// TIA Portal V17 export
// export: Created 2025-03-07T09:19:26.4228725Z, ExportSetting WithDefaults, DisplayName Totally Integrated Automation Portal, DisplayVersion V17 Update 8, DisplayName TIA Portal Openness, DisplayVersion V17 Update 8, DisplayName TIA Portal Version Control Interface, DisplayVersion V17, DisplayName SINAMICS Startdrive Advanced, DisplayVersion V17 SP2, DisplayName SINAMICS Startdrive G110M, G120, G120C, G120D, G120P, G115D, DisplayVersion V17 SP2, DisplayName SINAMICS Startdrive G130, G150, S120, S150, SINAMICS MV, S210, DisplayVersion V17 SP2, DisplayName STEP 7 Professional, DisplayVersion V17 Update 8, DisplayName SINUMERIK ONE STEP 7 Toolbox, DisplayVersion V17 Update 12, DisplayName SINUMERIK 840D sl STEP 7 Toolbox, DisplayVersion V17 Update 12, DisplayName STEP 7 Safety, DisplayVersion V17 Update 6, DisplayName WinCC Advanced, DisplayVersion V17 Update 8
TYPE "LBP_typeConfigData"
TITLE = Configuration parameter / Parámetros de configuración / Konfigurationsparameter
// User data type for block LBP_ConfigData [DB7] / Tipo de dato de usuario para bloque LBP_ConfigData [DB7] / Anwender-Datentyp für Baustein LBP_ConfigData [DB7]
// stored: IsFailsafeCompliant false
   STRUCT
      MCPNum : Int;   // Eingänge beginnen hier / Inputs starting here / Entradas comienzan aquí
      MCP1In : Struct   // Zeiger / Pointer / Puntero
         DBNo : Word;
         Addr : DWord;
      END_STRUCT;
      MCP1Out : Struct   // Zeiger / Pointer / Puntero
         DBNo : Word;
         Addr : DWord;
      END_STRUCT;
      reservedByte14_25 : Array[14..25] of Byte;
      MCP1BusAdr : Int := 6;
      MCP1Timeout : S5Time := S5T#700MS;
      reservedByte30_31 : Array[30..31] of Byte;
      MCP2In : Struct   // Zeiger / Pointer / Puntero
         DBNo : Word;
         Addr : DWord;
      END_STRUCT;
      MCP2Out : Struct   // Zeiger / Pointer / Puntero
         DBNo : Word;
         Addr : DWord;
      END_STRUCT;
      reservedByte44_55 : Array[44..55] of Byte;
      MCP2BusAdr : Int;
      MCP2Timeout : S5Time := S5T#700MS;
      reservedByte60_61 : Array[60..61] of Byte;
      reservedBool62_0 : Bool;
      MCP1Stop : Bool;
      MCP2Stop : Bool;
      MCP1NotSend : Bool;
      MCP2NotSend : Bool;
      reservedBool62_5 : Bool;
      reservedBool62_6 : Bool;
      MCPBusType : Byte := BYTE#16#05;
      HTIf : Int;
      HTIn : Struct   // Zeiger / Pointer / Puntero
         DBNo : Word;
         Addr : DWord;
      END_STRUCT;
      HTOut : Struct   // Zeiger / Pointer / Puntero
         DBNo : Word;
         Addr : DWord;
      END_STRUCT;
      reservedByte78_95 : Array[78..95] of Byte;
      HTAdr : Int := 2;
      reservedByte98_107 : Array[98..107] of Byte;
      reservedBool108_0 : Bool;
      HTStop : Bool;
      HTNotSend : Bool;
      NCCyclTimeout : S5Time := S5T#200MS;
      NCRunupTimeout : S5Time := S5T#50S;
      ListMDecGrp : Int;
      reservedBool116_0 : Bool;
      MMCToIF : Bool := TRUE;
      HWheelMMC : Bool := TRUE;
      reservedBool116_3 : Bool;
      MCP_IF_TCS : Bool;
      ExtendChanAxMsg : Bool;
      HMIAxisSel : Bool;
      DeactivateCtrlEnergy : Bool;
      MsgUser : Int := 10;
      reservedBool120_0 : Bool;
      IRAuxfuT : Bool;
      IRAuxfuH : Bool;
      IRAuxfuE : Bool;
      UserVersion : Struct   // Zeiger / Pointer / Puntero
         DBNo : Word;
         Addr : DWord;
      END_STRUCT;
      OpKeyNum : Int;
      Op1KeyIn : Struct   // Zeiger / Pointer / Puntero
         DBNo : Word;
         Addr : DWord;
      END_STRUCT;
      Op1KeyOut : Struct   // Zeiger / Pointer / Puntero
         DBNo : Word;
         Addr : DWord;
      END_STRUCT;
      Op1KeyBusAdr : Int;
      Op2KeyIn : Struct   // Zeiger / Pointer / Puntero
         DBNo : Word;
         Addr : DWord;
      END_STRUCT;
      Op2KeyOut : Struct   // Zeiger / Pointer / Puntero
         DBNo : Word;
         Addr : DWord;
      END_STRUCT;
      Op2KeyBusAdr : Int;
      Op1KeyStop : Bool;
      Op2KeyStop : Bool;
      Op1KeyNotSend : Bool;
      Op2KeyNotSend : Bool;
      reservedByte159 : Byte;
      IdentMcpBusAdr : Int;
      IdentMcpProfilNo : Byte;
      IdentMcpBusType : Byte := BYTE#16#05;
      IdentMcpStrobe : Bool;
      MaxModeGroup : Int;   // Ausgänge beginnen hier / Outputs starting here / Salidas comienzan aquí
      MaxChan : Int;
      MaxAxis : Int;
      ActiveChan : Array[1..10] of Bool;
      ActiveAxis : Array[1..31] of Bool;
      MaxNumUserDataInt : Int;
      MaxNumUserDataHex : Int;
      MaxNumUserDataReal : Int;
      IdentMcpType : Byte;
      IdentMcpLengthIn : Byte;
      IdentMcpLengthOut : Byte;
      reservedByte188_199 : Array[188..199] of Byte;   // Statisch beginnt hier / Static starting here / Estático comienza aquí
      LBPVersionInfo : String[44];
      UserVersionInfo : String[44];
      GenerateAlarmMsgs : Struct
         NumActAlarmMsgs : UInt;
         Error : Bool;
         StatusID : UInt;
         Status : Word;
      END_STRUCT;
      OpUnitCommId : UInt := 1;   // ID für OpUnitComm / ID for OpUnitComm / ID para OpUnitComm
      OpUnitInterfaceId : HW_ANY := 262;   // Hardware-Kennung der Ethernet-Schnittstelle für OpUnitComm / Hardware identifier of Ethernet interface for OpUnitComm / Identificador de hardware para interfaz Ethernet para OpUnitComm
      MCP1ConnectionId : CONN_OUC := 1001;   // Verbindungskennung für MCP 1 / Connection identifier for MCP 1 / Identificador de conexión para MCP 1
      MCP2ConnectionId : CONN_OUC := 1002;   // Verbindungskennung für MCP 2 / Connection identifier for MCP 2 / Identificador de conexión para MCP 2
      HTConnectionId : CONN_OUC := 1003;   // Verbindungskennung für Handbediengerät / Connection identifier for handheld unit / Identificador de conexión para mando simplificado
      Op1KeyConnectionId : CONN_OUC := 1004;   // Verbindungskennung für Direct Key 1 / Connection identifier for Direct Key 1 / Identificador de conexión para Direct Key 1
      Op2KeyConnectionId : CONN_OUC := 1005;   // Verbindungskennung für Direct Key 2 / Connection identifier for Direct Key 2 / Identificador de conexión para Direct Key 2
      IdentConnectionId : CONN_OUC := 1006;   // Verbindungskennung zur Identifikation / Connection identifier for identification / Identificador de conexión para identificación
      MCP1LocalUdpPort : UInt := 16001;   // Lokaler UDP-Port für MCP 1 / Local UDP port for MCP 1 / Puerto UDP local para MCP 1
      MCP2LocalUdpPort : UInt := 16002;   // Lokaler UDP-Port für MCP 2 / Local UDP port for MCP 2 / Puerto UDP local para MCP 2
      HTLocalUdpPort : UInt := 16003;   // Lokaler UDP-Port für Handbediengerät / Local UDP port for handheld unit / Puerto UDP local para mando simplificado
      Op1KeyLocalUdpPort : UInt := 16004;   // Lokaler UDP-Port für Direct Key 1 / Local UDP port for Direct Key 1 / Puerto UDP local para Direct Key 1
      Op2KeyLocalUdpPort : UInt := 16005;   // Lokaler UDP-Port für Direct Key 2 / Local UDP port for Direct Key 2 / Puerto UDP local para Direct Key 2
      IdentLocalUdpPort : UInt := 16006;   // Lokaler UDP-Port für Ident / Local UDP port for Ident / Puerto UDP local para ident
      MCP1Error : Bool;   // Fehler MCP 1 / Error MCP 1
      MCP1Status : Word;   // Fehler Information MCP 1 / Error information MCP 1 / Error información MCP 1
      MCP2Error : Bool;   // Fehler MCP 2 / Error MCP 2
      MCP2Status : Word;   // Fehler Information MCP 2 / Error information MCP 2 / Error información MCP 2
      HTError : Bool;   // Fehler Handbediengerät / Error handheld unit / Error mando simplificado
      HTStatus : Word;   // Fehler Information Handbediengerät / Error information handheld unit / Error información mando simplificado
      Op1KeyError : Bool;   // Fehler Direct Key 1 / Error Direct Key 1
      Op1KeyStatus : Word;   // Fehler Information Direct Key 1 / Error information Direct Key 1 / Error información Direct Key 1
      Op2KeyError : Bool;   // Fehler Direct Key 2 / Error Direct Key 2
      Op2KeyStatus : Word;   // Fehler Information Direct Key 2 / Error information Direct Key 2 / Error información Direct Key 2
      IdentError : Bool;   // Fehler Identifikation / Error identification / Error de identificación
      IdentStatus : Word;   // Fehler Information Identifikation / Error information Identification / Error información identificación
      MCP1Ready : Bool;   // MCP1 verbunden / MCP1 connected / MCP 1 conectado
      MCP2Ready : Bool;   // MCP2 verbunden / MCP2 connected / MCP 2 conectado
      HTReady : Bool;   // Handbediengerät verbunden / Handheld unit connected / Mando simplificado conectado
      Op1KeyReady : Bool;   // Direct Key 1 verbunden / Direct Key 1 connected / Direct Key 1 conectado
      Op2KeyReady : Bool;   // Direct Key 2 verbunden / Direct Key 2 connected / Direct Key 2 conectado
   END_STRUCT;
END_TYPE
